KUKA KRL program: 1.src, 1.dat

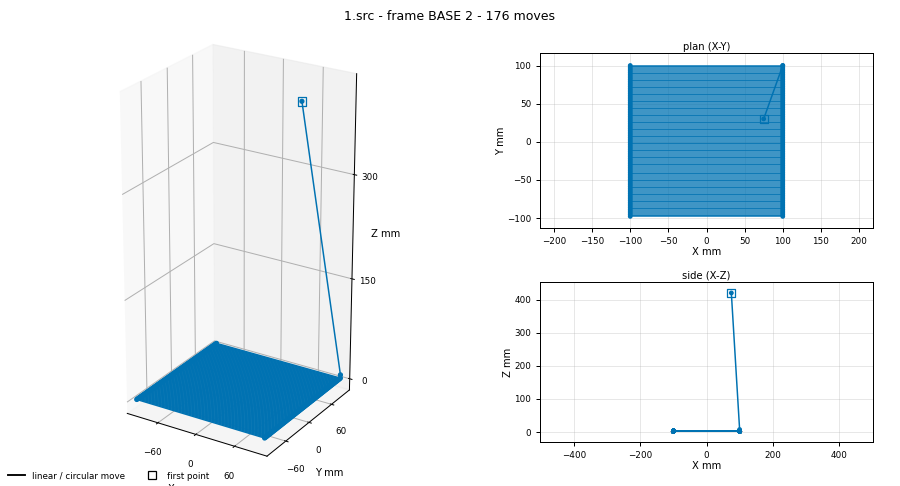
[picture p0: tool path of 1.src in frame BASE 2, 176 of 178 moves have a stored position in this frame; points joined in program order, loops and branches not executed]
--- 1.src ---
&ACCESS RVP
&PARAM TEMPLATE = C:\KRC\Roboter\Template\vorgabe
&PARAM EDITMASK = *
DEF 1( )
;FOLD INI;%{PE}%V3.2.0,%MKUKATPBASIS,%CINIT,%VCOMMON,%P
;FOLD BAS INI;%{E}%V3.2.0,%MKUKATPBASIS,%CINIT,%VINIT,%P
GLOBAL INTERRUPT DECL 3 WHEN $STOPMESS==TRUE DO IR_STOPM ( )
INTERRUPT ON 3
BAS (#INITMOV,0 )
;ENDFOLD (BAS INI)
;FOLD A20 INI;%{E}%V3.2.0,%MKUKATPA20,%CINIT,%VINIT,%P
IF ARC20==TRUE THEN
A20 (ARC_INI)
INTERRUPT DECL 6 WHEN $CYCFLAG[3]==FALSE DO A20(TECH_STOP2)
ENDIF
;ENDFOLD (A20 INI)
;FOLD A10 INI;%{E}%V3.2.0,%MKUKATPARC,%CINIT,%VINIT,%P
IF A10_OPTION==#ACTIVE THEN
INTERRUPT DECL 4 WHEN $CYCFLAG[2]==FALSE DO A10 (#APPL_ERROR)
INTERRUPT DECL 7 WHEN A_ARC_SWI==#ACTIVE DO A10 (#ARC_SEAM)
INTERRUPT DECL 5 WHEN A_FLY_ARC==TRUE DO A10 (#HPU_ARC)
INTERRUPT  ON 5
A10_INI ( )
ENDIF
;ENDFOLD (A10 INI)
;FOLD GRIPPER INI;%{E}%V3.2.0,%MKUKATPGRIPPER,%CINIT,%VINIT,%P
USER_GRP(0,DUMMY,DUMMY,GDEFAULT)
;ENDFOLD (GRIPPER INI)
;FOLD SPOT INI;%{E}%V3.2.0,%MKUKATPSPOT,%CINIT,%VINIT,%P
USERSPOT(#INIT)
;ENDFOLD (SPOT INI)
;FOLD TOUCHSENSE INI;%{E}%V3.2.0,%MKUKATPTS,%CINIT,%VINIT,%P
IF H70_OPTION THEN
INTERRUPT DECL 15 WHEN $MEAS_PULSE[TOUCH_I[TOUCH_ACTIVE].IN_NR] DO H70 (6,CD0 )
INTERRUPT DECL 16 WHEN $ZERO_MOVE DO H70 (7,CD0 )
INTERRUPT DECL 17 WHEN $TECHPAR_C[FG_TOUCH,8]>0.5 DO H70 (8,CD0)
H70 (1,CD0 )
ENDIF
;ENDFOLD (TOUCHSENSE INI)
;FOLD USER INI;%{E}%V3.2.0,%MKUKATPUSER,%CINIT,%VINIT,%P
;Make your modifications here
;ENDFOLD (USER INI)
;ENDFOLD (INI)
; SPEED PTP FOR AXIS
$VEL_AXIS[1] = 15
$VEL_AXIS[2] = 15
$VEL_AXIS[3] = 15
$VEL_AXIS[4] = 15
$VEL_AXIS[5] = 15
$VEL_AXIS[6] = 15
;SMOOTHNESS
$APO.CDIS = 2
;ADVANCE
$ADVANCE = 3
;SET TOOL AND BASE
$TOOL = TOOL_DATA[3]
$BASE = BASE_DATA[2]
;HOME
;FOLD PTP HOME Vel=10% DEFAULT
$BWDSTART=FALSE
$H_POS=XHOME
PDAT_ACT=PDEFAULT
FDAT_ACT=FHOME
BAS(#PTP_DAT )
BAS (#VEL_PTP,10 )
PTP XHOME
;ENDFOLD
;USER PROGRAM
;SPEED $VEL.CP
$VEL.CP=0.045
; OUT[TEMP] = 200
; OUT[vent] = 1
; OUT[RPM] = 45
; USER POSES CALLS
PTP {X 75, Y 30, Z 420, A 0, B 90, C 0}
; USER POSES CALLS
LIN {X 100.0, Y 100.0, Z 7.5, A 0, B 90, C 0} C_DIS
WAIT SEC 1
$OUT[1] = TRUE
LIN {X 100.0, Y 100.0, Z 2.5, A 0, B 90, C 0} C_DIS
LIN {X -100.0, Y 100.0, Z 2.5, A 0, B 90, C 0} C_DIS
LIN {X -100.0, Y 97.7, Z 2.5, A 0, B 90, C 0} C_DIS
LIN {X 100.0, Y 97.7, Z 2.5, A 0, B 90, C 0} C_DIS
LIN {X 100.0, Y 95.4, Z 2.5, A 0, B 90, C 0} C_DIS
LIN {X -100.0, Y 95.4, Z 2.5, A 0, B 90, C 0} C_DIS
LIN {X -100.0, Y 93.1, Z 2.5, A 0, B 90, C 0} C_DIS
LIN {X 100.0, Y 93.1, Z 2.5, A 0, B 90, C 0} C_DIS
LIN {X 100.0, Y 90.8, Z 2.5, A 0, B 90, C 0} C_DIS
LIN {X -100.0, Y 90.8, Z 2.5, A 0, B 90, C 0} C_DIS
LIN {X -100.0, Y 88.5, Z 2.5, A 0, B 90, C 0} C_DIS
LIN {X 100.0, Y 88.5, Z 2.5, A 0, B 90, C 0} C_DIS
LIN {X 100.0, Y 86.2, Z 2.5, A 0, B 90, C 0} C_DIS
LIN {X -100.0, Y 86.2, Z 2.5, A 0, B 90, C 0} C_DIS
LIN {X -100.0, Y 83.9, Z 2.5, A 0, B 90, C 0} C_DIS
LIN {X 100.0, Y 83.9, Z 2.5, A 0, B 90, C 0} C_DIS
LIN {X 100.0, Y 81.6, Z 2.5, A 0, B 90, C 0} C_DIS
LIN {X -100.0, Y 81.6, Z 2.5, A 0, B 90, C 0} C_DIS
LIN {X -100.0, Y 79.3, Z 2.5, A 0, B 90, C 0} C_DIS
LIN {X 100.0, Y 79.3, Z 2.5, A 0, B 90, C 0} C_DIS
LIN {X 100.0, Y 77.0, Z 2.5, A 0, B 90, C 0} C_DIS
LIN {X -100.0, Y 77.0, Z 2.5, A 0, B 90, C 0} C_DIS
LIN {X -100.0, Y 74.7, Z 2.5, A 0, B 90, C 0} C_DIS
LIN {X 100.0, Y 74.7, Z 2.5, A 0, B 90, C 0} C_DIS
LIN {X 100.0, Y 72.4, Z 2.5, A 0, B 90, C 0} C_DIS
LIN {X -100.0, Y 72.4, Z 2.5, A 0, B 90, C 0} C_DIS
LIN {X -100.0, Y 70.1, Z 2.5, A 0, B 90, C 0} C_DIS
LIN {X 100.0, Y 70.1, Z 2.5, A 0, B 90, C 0} C_DIS
LIN {X 100.0, Y 67.8, Z 2.5, A 0, B 90, C 0} C_DIS
LIN {X -100.0, Y 67.8, Z 2.5, A 0, B 90, C 0} C_DIS
LIN {X -100.0, Y 65.5, Z 2.5, A 0, B 90, C 0} C_DIS
LIN {X 100.0, Y 65.5, Z 2.5, A 0, B 90, C 0} C_DIS
LIN {X 100.0, Y 63.2, Z 2.5, A 0, B 90, C 0} C_DIS
LIN {X -100.0, Y 63.2, Z 2.5, A 0, B 90, C 0} C_DIS
LIN {X -100.0, Y 60.9, Z 2.5, A 0, B 90, C 0} C_DIS
LIN {X 100.0, Y 60.9, Z 2.5, A 0, B 90, C 0} C_DIS
LIN {X 100.0, Y 58.6, Z 2.5, A 0, B 90, C 0} C_DIS
LIN {X -100.0, Y 58.6, Z 2.5, A 0, B 90, C 0} C_DIS
LIN {X -100.0, Y 56.3, Z 2.5, A 0, B 90, C 0} C_DIS
LIN {X 100.0, Y 56.3, Z 2.5, A 0, B 90, C 0} C_DIS
LIN {X 100.0, Y 54.0, Z 2.5, A 0, B 90, C 0} C_DIS
LIN {X -100.0, Y 54.0, Z 2.5, A 0, B 90, C 0} C_DIS
LIN {X -100.0, Y 51.7, Z 2.5, A 0, B 90, C 0} C_DIS
LIN {X 100.0, Y 51.7, Z 2.5, A 0, B 90, C 0} C_DIS
LIN {X 100.0, Y 49.4, Z 2.5, A 0, B 90, C 0} C_DIS
LIN {X -100.0, Y 49.4, Z 2.5, A 0, B 90, C 0} C_DIS
LIN {X -100.0, Y 47.1, Z 2.5, A 0, B 90, C 0} C_DIS
LIN {X 100.0, Y 47.1, Z 2.5, A 0, B 90, C 0} C_DIS
LIN {X 100.0, Y 44.8, Z 2.5, A 0, B 90, C 0} C_DIS
LIN {X -100.0, Y 44.8, Z 2.5, A 0, B 90, C 0} C_DIS
LIN {X -100.0, Y 42.5, Z 2.5, A 0, B 90, C 0} C_DIS
LIN {X 100.0, Y 42.5, Z 2.5, A 0, B 90, C 0} C_DIS
LIN {X 100.0, Y 40.2, Z 2.5, A 0, B 90, C 0} C_DIS
LIN {X -100.0, Y 40.2, Z 2.5, A 0, B 90, C 0} C_DIS
LIN {X -100.0, Y 37.9, Z 2.5, A 0, B 90, C 0} C_DIS
LIN {X 100.0, Y 37.9, Z 2.5, A 0, B 90, C 0} C_DIS
LIN {X 100.0, Y 35.6, Z 2.5, A 0, B 90, C 0} C_DIS
LIN {X -100.0, Y 35.6, Z 2.5, A 0, B 90, C 0} C_DIS
LIN {X -100.0, Y 33.3, Z 2.5, A 0, B 90, C 0} C_DIS
LIN {X 100.0, Y 33.3, Z 2.5, A 0, B 90, C 0} C_DIS
LIN {X 100.0, Y 31.0, Z 2.5, A 0, B 90, C 0} C_DIS
LIN {X -100.0, Y 31.0, Z 2.5, A 0, B 90, C 0} C_DIS
LIN {X -100.0, Y 28.7, Z 2.5, A 0, B 90, C 0} C_DIS
LIN {X 100.0, Y 28.7, Z 2.5, A 0, B 90, C 0} C_DIS
LIN {X 100.0, Y 26.4, Z 2.5, A 0, B 90, C 0} C_DIS
LIN {X -100.0, Y 26.4, Z 2.5, A 0, B 90, C 0} C_DIS
LIN {X -100.0, Y 24.1, Z 2.5, A 0, B 90, C 0} C_DIS
LIN {X 100.0, Y 24.1, Z 2.5, A 0, B 90, C 0} C_DIS
LIN {X 100.0, Y 21.8, Z 2.5, A 0, B 90, C 0} C_DIS
LIN {X -100.0, Y 21.8, Z 2.5, A 0, B 90, C 0} C_DIS
LIN {X -100.0, Y 19.5, Z 2.5, A 0, B 90, C 0} C_DIS
LIN {X 100.0, Y 19.5, Z 2.5, A 0, B 90, C 0} C_DIS
LIN {X 100.0, Y 17.2, Z 2.5, A 0, B 90, C 0} C_DIS
LIN {X -100.0, Y 17.2, Z 2.5, A 0, B 90, C 0} C_DIS
LIN {X -100.0, Y 14.9, Z 2.5, A 0, B 90, C 0} C_DIS
LIN {X 100.0, Y 14.9, Z 2.5, A 0, B 90, C 0} C_DIS
LIN {X 100.0, Y 12.6, Z 2.5, A 0, B 90, C 0} C_DIS
LIN {X -100.0, Y 12.6, Z 2.5, A 0, B 90, C 0} C_DIS
LIN {X -100.0, Y 10.3, Z 2.5, A 0, B 90, C 0} C_DIS
LIN {X 100.0, Y 10.3, Z 2.5, A 0, B 90, C 0} C_DIS
LIN {X 100.0, Y 8.0, Z 2.5, A 0, B 90, C 0} C_DIS
LIN {X -100.0, Y 8.0, Z 2.5, A 0, B 90, C 0} C_DIS
LIN {X -100.0, Y 5.7, Z 2.5, A 0, B 90, C 0} C_DIS
LIN {X 100.0, Y 5.7, Z 2.5, A 0, B 90, C 0} C_DIS
LIN {X 100.0, Y 3.4, Z 2.5, A 0, B 90, C 0} C_DIS
LIN {X -100.0, Y 3.4, Z 2.5, A 0, B 90, C 0} C_DIS
LIN {X -100.0, Y 1.1, Z 2.5, A 0, B 90, C 0} C_DIS
LIN {X 100.0, Y 1.1, Z 2.5, A 0, B 90, C 0} C_DIS
LIN {X 100.0, Y -1.2, Z 2.5, A 0, B 90, C 0} C_DIS
LIN {X -100.0, Y -1.2, Z 2.5, A 0, B 90, C 0} C_DIS
LIN {X -100.0, Y -3.5, Z 2.5, A 0, B 90, C 0} C_DIS
LIN {X 100.0, Y -3.5, Z 2.5, A 0, B 90, C 0} C_DIS
LIN {X 100.0, Y -5.8, Z 2.5, A 0, B 90, C 0} C_DIS
LIN {X -100.0, Y -5.8, Z 2.5, A 0, B 90, C 0} C_DIS
LIN {X -100.0, Y -8.1, Z 2.5, A 0, B 90, C 0} C_DIS
LIN {X 100.0, Y -8.1, Z 2.5, A 0, B 90, C 0} C_DIS
LIN {X 100.0, Y -10.4, Z 2.5, A 0, B 90, C 0} C_DIS
LIN {X -100.0, Y -10.4, Z 2.5, A 0, B 90, C 0} C_DIS
LIN {X -100.0, Y -12.7, Z 2.5, A 0, B 90, C 0} C_DIS
LIN {X 100.0, Y -12.7, Z 2.5, A 0, B 90, C 0} C_DIS
LIN {X 100.0, Y -15.0, Z 2.5, A 0, B 90, C 0} C_DIS
LIN {X -100.0, Y -15.0, Z 2.5, A 0, B 90, C 0} C_DIS
LIN {X -100.0, Y -17.3, Z 2.5, A 0, B 90, C 0} C_DIS
LIN {X 100.0, Y -17.3, Z 2.5, A 0, B 90, C 0} C_DIS
LIN {X 100.0, Y -19.6, Z 2.5, A 0, B 90, C 0} C_DIS
LIN {X -100.0, Y -19.6, Z 2.5, A 0, B 90, C 0} C_DIS
LIN {X -100.0, Y -21.9, Z 2.5, A 0, B 90, C 0} C_DIS
LIN {X 100.0, Y -21.9, Z 2.5, A 0, B 90, C 0} C_DIS
LIN {X 100.0, Y -24.2, Z 2.5, A 0, B 90, C 0} C_DIS
LIN {X -100.0, Y -24.2, Z 2.5, A 0, B 90, C 0} C_DIS
LIN {X -100.0, Y -26.5, Z 2.5, A 0, B 90, C 0} C_DIS
LIN {X 100.0, Y -26.5, Z 2.5, A 0, B 90, C 0} C_DIS
LIN {X 100.0, Y -28.8, Z 2.5, A 0, B 90, C 0} C_DIS
LIN {X -100.0, Y -28.8, Z 2.5, A 0, B 90, C 0} C_DIS
LIN {X -100.0, Y -31.1, Z 2.5, A 0, B 90, C 0} C_DIS
LIN {X 100.0, Y -31.1, Z 2.5, A 0, B 90, C 0} C_DIS
LIN {X 100.0, Y -33.4, Z 2.5, A 0, B 90, C 0} C_DIS
LIN {X -100.0, Y -33.4, Z 2.5, A 0, B 90, C 0} C_DIS
LIN {X -100.0, Y -35.7, Z 2.5, A 0, B 90, C 0} C_DIS
LIN {X 100.0, Y -35.7, Z 2.5, A 0, B 90, C 0} C_DIS
LIN {X 100.0, Y -38.0, Z 2.5, A 0, B 90, C 0} C_DIS
LIN {X -100.0, Y -38.0, Z 2.5, A 0, B 90, C 0} C_DIS
LIN {X -100.0, Y -40.3, Z 2.5, A 0, B 90, C 0} C_DIS
LIN {X 100.0, Y -40.3, Z 2.5, A 0, B 90, C 0} C_DIS
LIN {X 100.0, Y -42.6, Z 2.5, A 0, B 90, C 0} C_DIS
LIN {X -100.0, Y -42.6, Z 2.5, A 0, B 90, C 0} C_DIS
LIN {X -100.0, Y -44.9, Z 2.5, A 0, B 90, C 0} C_DIS
LIN {X 100.0, Y -44.9, Z 2.5, A 0, B 90, C 0} C_DIS
LIN {X 100.0, Y -47.2, Z 2.5, A 0, B 90, C 0} C_DIS
LIN {X -100.0, Y -47.2, Z 2.5, A 0, B 90, C 0} C_DIS
LIN {X -100.0, Y -49.5, Z 2.5, A 0, B 90, C 0} C_DIS
LIN {X 100.0, Y -49.5, Z 2.5, A 0, B 90, C 0} C_DIS
LIN {X 100.0, Y -51.8, Z 2.5, A 0, B 90, C 0} C_DIS
LIN {X -100.0, Y -51.8, Z 2.5, A 0, B 90, C 0} C_DIS
LIN {X -100.0, Y -54.1, Z 2.5, A 0, B 90, C 0} C_DIS
LIN {X 100.0, Y -54.1, Z 2.5, A 0, B 90, C 0} C_DIS
LIN {X 100.0, Y -56.4, Z 2.5, A 0, B 90, C 0} C_DIS
LIN {X -100.0, Y -56.4, Z 2.5, A 0, B 90, C 0} C_DIS
LIN {X -100.0, Y -58.7, Z 2.5, A 0, B 90, C 0} C_DIS
LIN {X 100.0, Y -58.7, Z 2.5, A 0, B 90, C 0} C_DIS
LIN {X 100.0, Y -61.0, Z 2.5, A 0, B 90, C 0} C_DIS
LIN {X -100.0, Y -61.0, Z 2.5, A 0, B 90, C 0} C_DIS
LIN {X -100.0, Y -63.3, Z 2.5, A 0, B 90, C 0} C_DIS
LIN {X 100.0, Y -63.3, Z 2.5, A 0, B 90, C 0} C_DIS
LIN {X 100.0, Y -65.6, Z 2.5, A 0, B 90, C 0} C_DIS
LIN {X -100.0, Y -65.6, Z 2.5, A 0, B 90, C 0} C_DIS
LIN {X -100.0, Y -67.9, Z 2.5, A 0, B 90, C 0} C_DIS
LIN {X 100.0, Y -67.9, Z 2.5, A 0, B 90, C 0} C_DIS
LIN {X 100.0, Y -70.2, Z 2.5, A 0, B 90, C 0} C_DIS
LIN {X -100.0, Y -70.2, Z 2.5, A 0, B 90, C 0} C_DIS
LIN {X -100.0, Y -72.5, Z 2.5, A 0, B 90, C 0} C_DIS
LIN {X 100.0, Y -72.5, Z 2.5, A 0, B 90, C 0} C_DIS
LIN {X 100.0, Y -74.8, Z 2.5, A 0, B 90, C 0} C_DIS
LIN {X -100.0, Y -74.8, Z 2.5, A 0, B 90, C 0} C_DIS
LIN {X -100.0, Y -77.1, Z 2.5, A 0, B 90, C 0} C_DIS
LIN {X 100.0, Y -77.1, Z 2.5, A 0, B 90, C 0} C_DIS
LIN {X 100.0, Y -79.4, Z 2.5, A 0, B 90, C 0} C_DIS
LIN {X -100.0, Y -79.4, Z 2.5, A 0, B 90, C 0} C_DIS
LIN {X -100.0, Y -81.7, Z 2.5, A 0, B 90, C 0} C_DIS
LIN {X 100.0, Y -81.7, Z 2.5, A 0, B 90, C 0} C_DIS
LIN {X 100.0, Y -84.0, Z 2.5, A 0, B 90, C 0} C_DIS
LIN {X -100.0, Y -84.0, Z 2.5, A 0, B 90, C 0} C_DIS
LIN {X -100.0, Y -86.3, Z 2.5, A 0, B 90, C 0} C_DIS
LIN {X 100.0, Y -86.3, Z 2.5, A 0, B 90, C 0} C_DIS
LIN {X 100.0, Y -88.6, Z 2.5, A 0, B 90, C 0} C_DIS
LIN {X -100.0, Y -88.6, Z 2.5, A 0, B 90, C 0} C_DIS
LIN {X -100.0, Y -90.9, Z 2.5, A 0, B 90, C 0} C_DIS
LIN {X 100.0, Y -90.9, Z 2.5, A 0, B 90, C 0} C_DIS
LIN {X 100.0, Y -93.2, Z 2.5, A 0, B 90, C 0} C_DIS
LIN {X -100.0, Y -93.2, Z 2.5, A 0, B 90, C 0} C_DIS
LIN {X -100.0, Y -95.5, Z 2.5, A 0, B 90, C 0} C_DIS
LIN {X 100.0, Y -95.5, Z 2.5, A 0, B 90, C 0} C_DIS
LIN {X 100.0, Y -97.8, Z 2.5, A 0, B 90, C 0} C_DIS
LIN {X -100.0, Y -97.8, Z 2.5, A 0, B 90, C 0} C_DIS
$OUT[1] = FALSE

;Wait for
; END POSITION FOR
;END USER CODE
;HOME
;FOLD PTP HOME Vel=10% DEFAULT
$BWDSTART=FALSE
$H_POS=XHOME
PDAT_ACT=PDEFAULT
FDAT_ACT=FHOME
BAS(#PTP_DAT )
BAS (#VEL_PTP,10 )
PTP XHOME
;ENDFOLD
END

--- 1.dat ---
DEFDAT 1()
ENDDAT
